FUNCTION_BLOCK FB_StableValue //stabiler wert
VAR_INPUT
	fValue		: LREAL;
	iPrecision	: INT;
	bRound		: BOOL;
	tStabileTon	: TIME := T#50MS;
	tStabileTof	: TIME := T#20MS;
END_VAR
VAR_OUTPUT
	sValue				: STRING;
	fValueFmt			: LREAL;
	bStabileValue		: BOOL;
	bStabileValueTout	: BOOL;
END_VAR
VAR
	fTempValue	: LREAL;
	tonStabile	: TON;
	tofStabile	: TOf;
END_VAR


sValue := LREAL_TO_FMTSTR(fValue,iPrecision,bRound);
fValueFmt := TO_LREAL(sValue);

IF (fValueFmt <> fTempValue) THEN
	fTempValue := fValueFmt;
END_IF
bStabileValue := (fValueFmt = fTempValue);

tonStabile.IN := bStabileValue;
tonStabile.PT := tStabileTon;
tonStabile();

tofStabile.IN := tonStabile.Q;
tofStabile.PT := tStabileTof;
tofStabile();

bStabileValueTout := tofStabile.Q;

END_FUNCTION_BLOCK

(* stored: Version 1.1.0.1, ProductVersion 3.1.4024.11
   POU FB_StableValue: Id {b6bc1479-e54d-4bb2-8207-1bfa2cdf7f2b}, SpecialFunc None *)
